// TIA Portal V18 export
FUNCTION_BLOCK "MES Check_fb"   // FB110, LAD
{ S7_Optimized_Access := 'TRUE' }
// stored: AutoNumber false, MemoryReserve 100, SetENOAutomatically false
   VAR_INPUT
      i_AlwaysTrue : Bool;
      i_MESOnlineOffline : Bool;
      i_CheckRequest : Bool;
      i_ResultRequest : Bool;
      i_Reset : Bool;
      i_CheckTimeOut : DInt := 10000;
      i_ResultTimeOut : DInt := 10000;
      i_Status : Int;
   END_VAR
   VAR_OUTPUT
      o_CheckTimeOut : Bool;
      o_ResultTimeOut : Bool;
   END_VAR
   VAR_IN_OUT
      ioPLC_MESCheckReq : Bool;
      ioPLC_MESResultReq : Bool;
      ioMES_PLCChecOK : Bool;
      ioMES_PLCChecNG : Bool;
      ioMES_PLCChecDone : Bool;
      ioMES_PLCResultOK : Bool;
      ioMES_PLCResultNG : Bool;
      ioMES_PLCResultDone : Bool;
      ioProductStatus : Int;
   END_VAR
   VAR
      CheckStep : Int;
      ResultStep : Int;
      CheckTimeOut : TON_TIME;
      ResultTimeOut { S7_SetPoint := 'True'} : TON_TIME;
      Pls : Array[0..20] of Bool;
   END_VAR
   VAR_TEMP   // added for the SCL form of the ladder/FBD networks
      _w1 : Bool;
      _w2 : Bool;
      _w3 : Bool;
      _w4 : Bool;
      _w5 : Bool;
      _w6 : Bool;
      _w7 : Bool;
   END_VAR
BEGIN

REGION Network 1: MES Check In Start
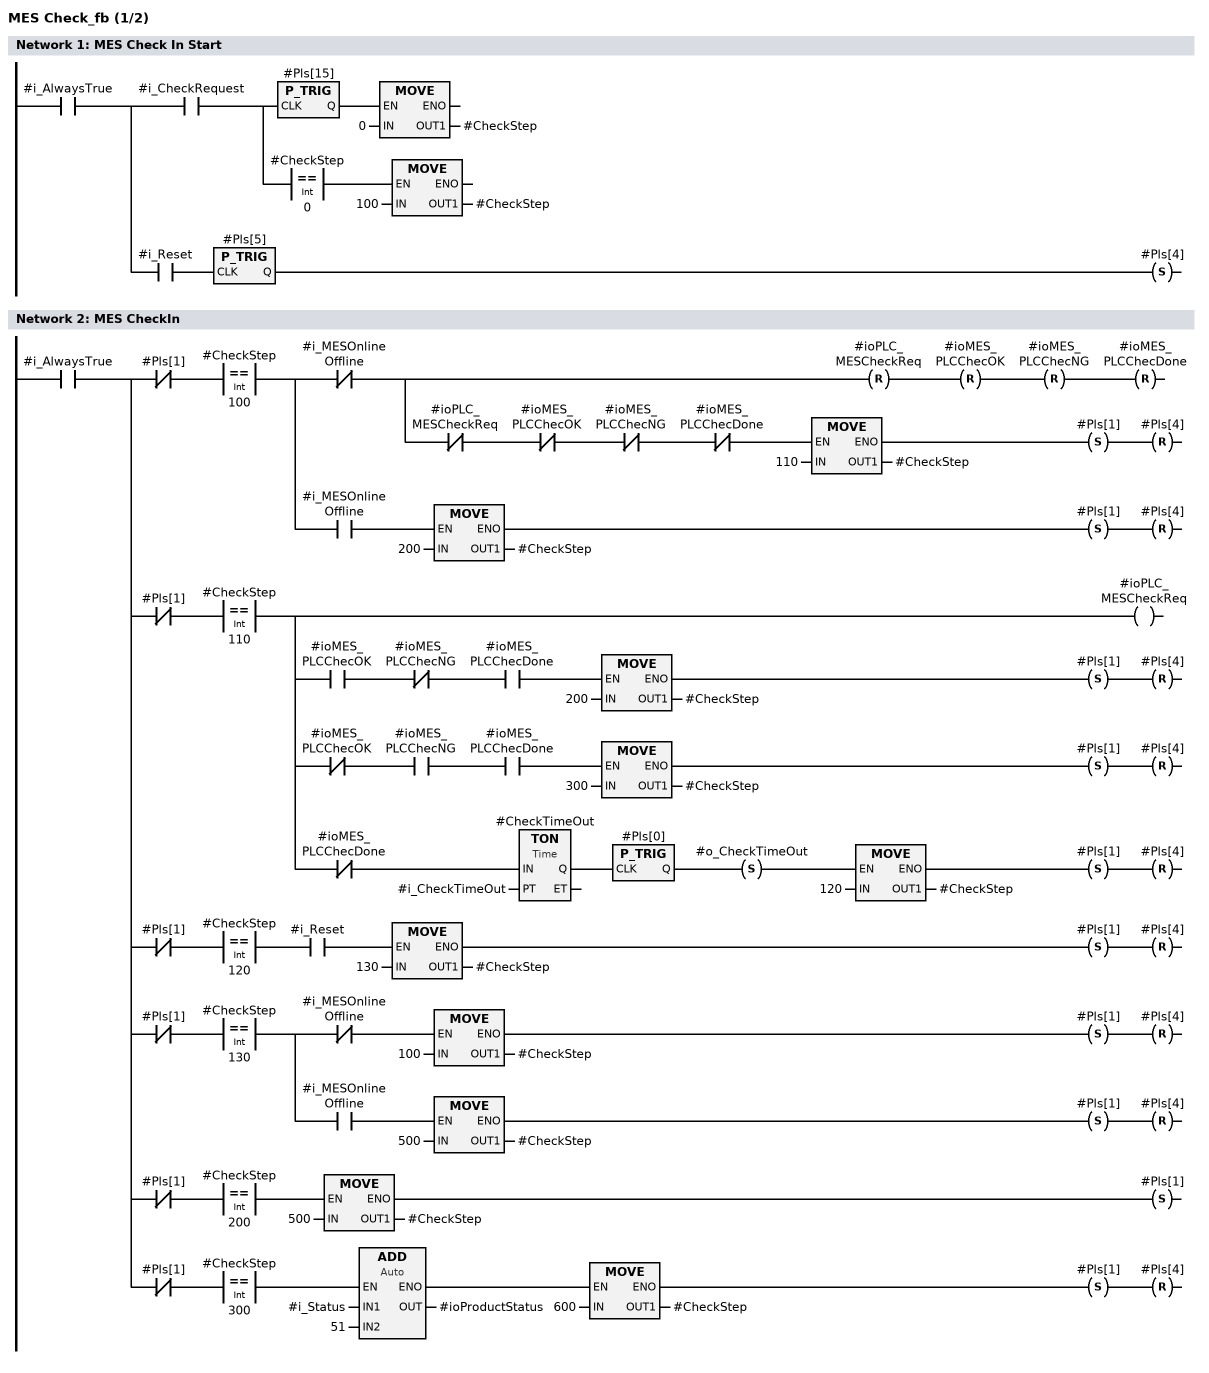
   RUNG wire#powerrail
      Contact( #i_AlwaysTrue )
      wire#w1
      Contact( #i_CheckRequest )
      wire#w2
      P_Trig( #Pls[15] )
      Move(in := 0, out1 => #CheckStep)
   END_RUNG
   RUNG wire#w2
      { S7_Templates := "SrcType := Int" } EQ_Contact(in1 := #CheckStep, in2 := 0)
      Move(in := 100, out1 => #CheckStep)
   END_RUNG
   RUNG wire#w1
      Contact( #i_Reset )
      P_Trig( #Pls[5] )
      S_Coil( #Pls[4] )
   END_RUNG
   // the same network as SCL:
   #_w1 := #i_AlwaysTrue AND #i_CheckRequest;
   #_w2 := #_w1 AND NOT #Pls[15];   // rising edge
   #Pls[15] := #_w1;
   IF #_w2 THEN #CheckStep := 0; END_IF;
   IF #_w1 AND (#CheckStep = 0) THEN #CheckStep := 100; END_IF;
   #_w3 := #i_AlwaysTrue AND #i_Reset;
   #_w4 := #_w3 AND NOT #Pls[5];   // rising edge
   #Pls[5] := #_w3;
   IF #_w4 THEN #Pls[4] := TRUE; END_IF;
END_REGION

REGION Network 2: MES CheckIn
   RUNG wire#powerrail
      Contact( #i_AlwaysTrue )
      wire#w1
      I_Contact( #Pls[1] )
      { S7_Templates := "SrcType := Int" } EQ_Contact(in1 := #CheckStep, in2 := 100)
      wire#w2
      I_Contact( #i_MESOnlineOffline )
      wire#w3
      R_Coil( #ioPLC_MESCheckReq )
      R_Coil( #ioMES_PLCChecOK )
      R_Coil( #ioMES_PLCChecNG )
      R_Coil( #ioMES_PLCChecDone )
   END_RUNG
   RUNG wire#w3
      I_Contact( #ioPLC_MESCheckReq )
      I_Contact( #ioMES_PLCChecOK )
      I_Contact( #ioMES_PLCChecNG )
      I_Contact( #ioMES_PLCChecDone )
      Move(in := 110, out1 => #CheckStep)
      S_Coil( #Pls[1] )
      R_Coil( #Pls[4] )
   END_RUNG
   RUNG wire#w2
      Contact( #i_MESOnlineOffline )
      Move(in := 200, out1 => #CheckStep)
      S_Coil( #Pls[1] )
      R_Coil( #Pls[4] )
   END_RUNG
   RUNG wire#w1
      I_Contact( #Pls[1] )
      { S7_Templates := "SrcType := Int" } EQ_Contact(in1 := #CheckStep, in2 := 110)
      wire#w4
      Coil( #ioPLC_MESCheckReq )
   END_RUNG
   RUNG wire#w4
      Contact( #ioMES_PLCChecOK )
      I_Contact( #ioMES_PLCChecNG )
      Contact( #ioMES_PLCChecDone )
      Move(in := 200, out1 => #CheckStep)
      S_Coil( #Pls[1] )
      R_Coil( #Pls[4] )
   END_RUNG
   RUNG wire#w4
      I_Contact( #ioMES_PLCChecOK )
      Contact( #ioMES_PLCChecNG )
      Contact( #ioMES_PLCChecDone )
      Move(in := 300, out1 => #CheckStep)
      S_Coil( #Pls[1] )
      R_Coil( #Pls[4] )
   END_RUNG
   RUNG wire#w4
      I_Contact( #ioMES_PLCChecDone )
      { S7_Templates := "time_type := Time" } #CheckTimeOut.TON(pt := #i_CheckTimeOut, et =>)
      P_Trig( #Pls[0] )
      S_Coil( #o_CheckTimeOut )
      Move(in := 120, out1 => #CheckStep)
      S_Coil( #Pls[1] )
      R_Coil( #Pls[4] )
   END_RUNG
   RUNG wire#w1
      I_Contact( #Pls[1] )
      { S7_Templates := "SrcType := Int" } EQ_Contact(in1 := #CheckStep, in2 := 120)
      Contact( #i_Reset )
      Move(in := 130, out1 => #CheckStep)
      S_Coil( #Pls[1] )
      R_Coil( #Pls[4] )
   END_RUNG
   RUNG wire#w1
      I_Contact( #Pls[1] )
      { S7_Templates := "SrcType := Int" } EQ_Contact(in1 := #CheckStep, in2 := 130)
      wire#w5
      I_Contact( #i_MESOnlineOffline )
      Move(in := 100, out1 => #CheckStep)
      S_Coil( #Pls[1] )
      R_Coil( #Pls[4] )
   END_RUNG
   RUNG wire#w5
      Contact( #i_MESOnlineOffline )
      Move(in := 500, out1 => #CheckStep)
      S_Coil( #Pls[1] )
      R_Coil( #Pls[4] )
   END_RUNG
   RUNG wire#w1
      I_Contact( #Pls[1] )
      { S7_Templates := "SrcType := Int" } EQ_Contact(in1 := #CheckStep, in2 := 200)
      Move(in := 500, out1 => #CheckStep)
      S_Coil( #Pls[1] )
   END_RUNG
   RUNG wire#w1
      I_Contact( #Pls[1] )
      { S7_Templates := "SrcType := Int" } EQ_Contact(in1 := #CheckStep, in2 := 300)
      Add(in1 := #i_Status, in2 := 51, out => #ioProductStatus)
      Move(in := 600, out1 => #CheckStep)
      S_Coil( #Pls[1] )
      R_Coil( #Pls[4] )
   END_RUNG
   // the same network as SCL:
   #_w1 := #i_AlwaysTrue AND NOT #Pls[1] AND (#CheckStep = 100);
   #_w2 := #_w1 AND NOT #i_MESOnlineOffline;
   IF #_w2 THEN
       #ioPLC_MESCheckReq := FALSE;
       #ioMES_PLCChecOK := FALSE;
       #ioMES_PLCChecNG := FALSE;
       #ioMES_PLCChecDone := FALSE;
   END_IF;
   IF #_w2 AND NOT #ioPLC_MESCheckReq AND NOT #ioMES_PLCChecOK AND NOT #ioMES_PLCChecNG AND NOT #ioMES_PLCChecDone THEN
       #CheckStep := 110;
       #Pls[1] := TRUE;
       #Pls[4] := FALSE;
   END_IF;
   IF #_w1 AND #i_MESOnlineOffline THEN
       #CheckStep := 200;
       #Pls[1] := TRUE;
       #Pls[4] := FALSE;
   END_IF;
   #ioPLC_MESCheckReq := #i_AlwaysTrue AND NOT #Pls[1] AND (#CheckStep = 110);
   IF #ioPLC_MESCheckReq AND #ioMES_PLCChecOK AND NOT #ioMES_PLCChecNG AND #ioMES_PLCChecDone THEN
       #CheckStep := 200;
       #Pls[1] := TRUE;
       #Pls[4] := FALSE;
   END_IF;
   IF #ioPLC_MESCheckReq AND NOT #ioMES_PLCChecOK AND #ioMES_PLCChecNG AND #ioMES_PLCChecDone THEN
       #CheckStep := 300;
       #Pls[1] := TRUE;
       #Pls[4] := FALSE;
   END_IF;
   #CheckTimeOut(IN := #ioPLC_MESCheckReq AND NOT #ioMES_PLCChecDone, PT := #i_CheckTimeOut);   // TON
   #_w3 := #CheckTimeOut.Q AND NOT #Pls[0];   // rising edge
   #Pls[0] := #CheckTimeOut.Q;
   IF #_w3 THEN
       #o_CheckTimeOut := TRUE;
       #CheckStep := 120;
       #Pls[1] := TRUE;
       #Pls[4] := FALSE;
   END_IF;
   #_w4 := #i_AlwaysTrue AND NOT #Pls[1] AND (#CheckStep = 120) AND #i_Reset;
   IF #_w4 THEN
       #CheckStep := 130;
       #Pls[1] := TRUE;
       #Pls[4] := FALSE;
   END_IF;
   #_w5 := #i_AlwaysTrue AND NOT #Pls[1] AND (#CheckStep = 130);
   IF #_w5 AND NOT #i_MESOnlineOffline THEN
       #CheckStep := 100;
       #Pls[1] := TRUE;
       #Pls[4] := FALSE;
   END_IF;
   IF #_w5 AND #i_MESOnlineOffline THEN
       #CheckStep := 500;
       #Pls[1] := TRUE;
       #Pls[4] := FALSE;
   END_IF;
   #_w6 := #i_AlwaysTrue AND NOT #Pls[1] AND (#CheckStep = 200);
   IF #_w6 THEN
       #CheckStep := 500;
       #Pls[1] := TRUE;
   END_IF;
   IF #i_AlwaysTrue AND NOT #Pls[1] AND (#CheckStep = 300) THEN #ioProductStatus := #i_Status + 51; END_IF;
   #_w7 := #i_AlwaysTrue AND NOT #Pls[1] AND (#CheckStep = 300);
   IF #_w7 THEN
       #CheckStep := 600;
       #Pls[1] := TRUE;
       #Pls[4] := FALSE;
   END_IF;
END_REGION

REGION Network 4: MES Check Out Start
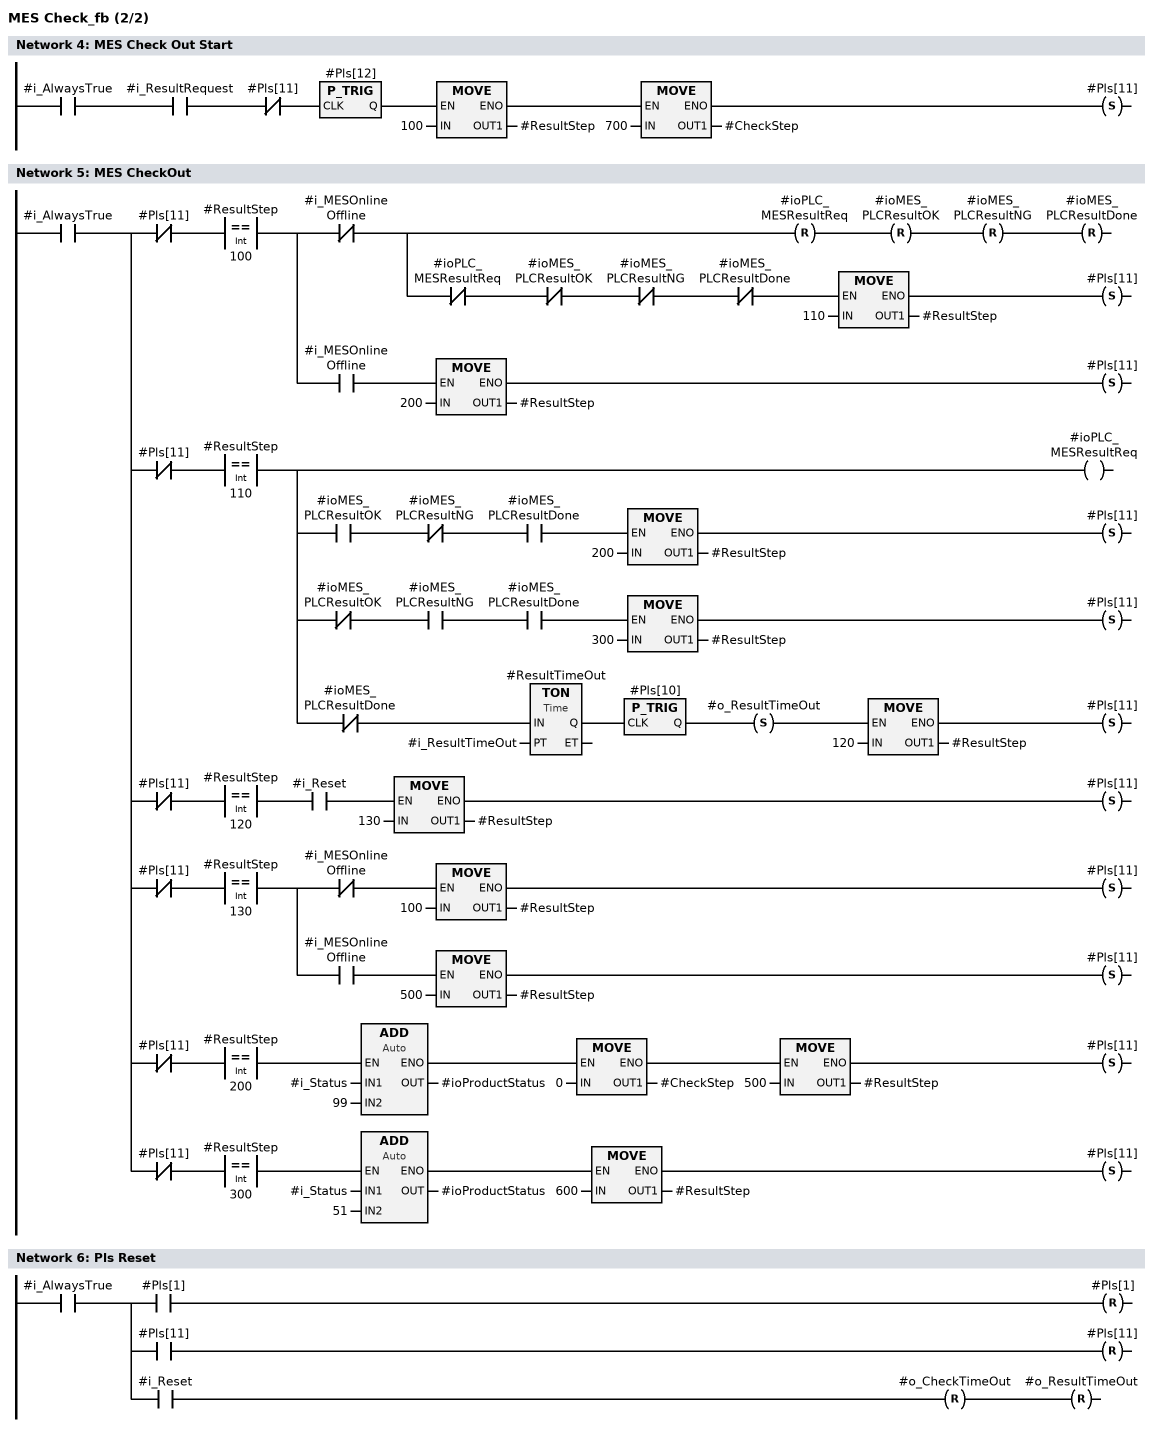
   RUNG wire#powerrail
      Contact( #i_AlwaysTrue )
      Contact( #i_ResultRequest )
      I_Contact( #Pls[11] )
      P_Trig( #Pls[12] )
      Move(in := 100, out1 => #ResultStep)
      Move(in := 700, out1 => #CheckStep)
      S_Coil( #Pls[11] )
   END_RUNG
   // the same network as SCL:
   #_w1 := #i_AlwaysTrue AND #i_ResultRequest AND NOT #Pls[11];
   #_w2 := #_w1 AND NOT #Pls[12];   // rising edge
   #Pls[12] := #_w1;
   IF #_w2 THEN
       #ResultStep := 100;
       #CheckStep := 700;
       #Pls[11] := TRUE;
   END_IF;
END_REGION

REGION Network 5: MES CheckOut
   RUNG wire#powerrail
      Contact( #i_AlwaysTrue )
      wire#w1
      I_Contact( #Pls[11] )
      { S7_Templates := "SrcType := Int" } EQ_Contact(in1 := #ResultStep, in2 := 100)
      wire#w2
      I_Contact( #i_MESOnlineOffline )
      wire#w3
      R_Coil( #ioPLC_MESResultReq )
      R_Coil( #ioMES_PLCResultOK )
      R_Coil( #ioMES_PLCResultNG )
      R_Coil( #ioMES_PLCResultDone )
   END_RUNG
   RUNG wire#w3
      I_Contact( #ioPLC_MESResultReq )
      I_Contact( #ioMES_PLCResultOK )
      I_Contact( #ioMES_PLCResultNG )
      I_Contact( #ioMES_PLCResultDone )
      Move(in := 110, out1 => #ResultStep)
      S_Coil( #Pls[11] )
   END_RUNG
   RUNG wire#w2
      Contact( #i_MESOnlineOffline )
      Move(in := 200, out1 => #ResultStep)
      S_Coil( #Pls[11] )
   END_RUNG
   RUNG wire#w1
      I_Contact( #Pls[11] )
      { S7_Templates := "SrcType := Int" } EQ_Contact(in1 := #ResultStep, in2 := 110)
      wire#w4
      Coil( #ioPLC_MESResultReq )
   END_RUNG
   RUNG wire#w4
      Contact( #ioMES_PLCResultOK )
      I_Contact( #ioMES_PLCResultNG )
      Contact( #ioMES_PLCResultDone )
      Move(in := 200, out1 => #ResultStep)
      S_Coil( #Pls[11] )
   END_RUNG
   RUNG wire#w4
      I_Contact( #ioMES_PLCResultOK )
      Contact( #ioMES_PLCResultNG )
      Contact( #ioMES_PLCResultDone )
      Move(in := 300, out1 => #ResultStep)
      S_Coil( #Pls[11] )
   END_RUNG
   RUNG wire#w4
      I_Contact( #ioMES_PLCResultDone )
      { S7_Templates := "time_type := Time" } #ResultTimeOut.TON(pt := #i_ResultTimeOut, et =>)
      P_Trig( #Pls[10] )
      S_Coil( #o_ResultTimeOut )
      Move(in := 120, out1 => #ResultStep)
      S_Coil( #Pls[11] )
   END_RUNG
   RUNG wire#w1
      I_Contact( #Pls[11] )
      { S7_Templates := "SrcType := Int" } EQ_Contact(in1 := #ResultStep, in2 := 120)
      Contact( #i_Reset )
      Move(in := 130, out1 => #ResultStep)
      S_Coil( #Pls[11] )
   END_RUNG
   RUNG wire#w1
      I_Contact( #Pls[11] )
      { S7_Templates := "SrcType := Int" } EQ_Contact(in1 := #ResultStep, in2 := 130)
      wire#w5
      I_Contact( #i_MESOnlineOffline )
      Move(in := 100, out1 => #ResultStep)
      S_Coil( #Pls[11] )
   END_RUNG
   RUNG wire#w5
      Contact( #i_MESOnlineOffline )
      Move(in := 500, out1 => #ResultStep)
      S_Coil( #Pls[11] )
   END_RUNG
   RUNG wire#w1
      I_Contact( #Pls[11] )
      { S7_Templates := "SrcType := Int" } EQ_Contact(in1 := #ResultStep, in2 := 200)
      Add(in1 := #i_Status, in2 := 99, out => #ioProductStatus)
      Move(in := 0, out1 => #CheckStep)
      Move(in := 500, out1 => #ResultStep)
      S_Coil( #Pls[11] )
   END_RUNG
   RUNG wire#w1
      I_Contact( #Pls[11] )
      { S7_Templates := "SrcType := Int" } EQ_Contact(in1 := #ResultStep, in2 := 300)
      Add(in1 := #i_Status, in2 := 51, out => #ioProductStatus)
      Move(in := 600, out1 => #ResultStep)
      S_Coil( #Pls[11] )
   END_RUNG
   // the same network as SCL:
   #_w1 := #i_AlwaysTrue AND NOT #Pls[11] AND (#ResultStep = 100);
   #_w2 := #_w1 AND NOT #i_MESOnlineOffline;
   IF #_w2 THEN
       #ioPLC_MESResultReq := FALSE;
       #ioMES_PLCResultOK := FALSE;
       #ioMES_PLCResultNG := FALSE;
       #ioMES_PLCResultDone := FALSE;
   END_IF;
   IF #_w2 AND NOT #ioPLC_MESResultReq AND NOT #ioMES_PLCResultOK AND NOT #ioMES_PLCResultNG AND NOT #ioMES_PLCResultDone THEN
       #ResultStep := 110;
       #Pls[11] := TRUE;
   END_IF;
   IF #_w1 AND #i_MESOnlineOffline THEN
       #ResultStep := 200;
       #Pls[11] := TRUE;
   END_IF;
   #ioPLC_MESResultReq := #i_AlwaysTrue AND NOT #Pls[11] AND (#ResultStep = 110);
   IF #ioPLC_MESResultReq AND #ioMES_PLCResultOK AND NOT #ioMES_PLCResultNG AND #ioMES_PLCResultDone THEN
       #ResultStep := 200;
       #Pls[11] := TRUE;
   END_IF;
   IF #ioPLC_MESResultReq AND NOT #ioMES_PLCResultOK AND #ioMES_PLCResultNG AND #ioMES_PLCResultDone THEN
       #ResultStep := 300;
       #Pls[11] := TRUE;
   END_IF;
   #ResultTimeOut(IN := #ioPLC_MESResultReq AND NOT #ioMES_PLCResultDone, PT := #i_ResultTimeOut);   // TON
   #_w3 := #ResultTimeOut.Q AND NOT #Pls[10];   // rising edge
   #Pls[10] := #ResultTimeOut.Q;
   IF #_w3 THEN
       #o_ResultTimeOut := TRUE;
       #ResultStep := 120;
       #Pls[11] := TRUE;
   END_IF;
   #_w4 := #i_AlwaysTrue AND NOT #Pls[11] AND (#ResultStep = 120) AND #i_Reset;
   IF #_w4 THEN
       #ResultStep := 130;
       #Pls[11] := TRUE;
   END_IF;
   #_w5 := #i_AlwaysTrue AND NOT #Pls[11] AND (#ResultStep = 130);
   IF #_w5 AND NOT #i_MESOnlineOffline THEN
       #ResultStep := 100;
       #Pls[11] := TRUE;
   END_IF;
   IF #_w5 AND #i_MESOnlineOffline THEN
       #ResultStep := 500;
       #Pls[11] := TRUE;
   END_IF;
   IF #i_AlwaysTrue AND NOT #Pls[11] AND (#ResultStep = 200) THEN
       #ioProductStatus := #i_Status + 99;
       #CheckStep := 0;
   END_IF;
   #_w6 := #i_AlwaysTrue AND NOT #Pls[11] AND (#ResultStep = 200);
   IF #_w6 THEN
       #ResultStep := 500;
       #Pls[11] := TRUE;
   END_IF;
   IF #i_AlwaysTrue AND NOT #Pls[11] AND (#ResultStep = 300) THEN #ioProductStatus := #i_Status + 51; END_IF;
   #_w7 := #i_AlwaysTrue AND NOT #Pls[11] AND (#ResultStep = 300);
   IF #_w7 THEN
       #ResultStep := 600;
       #Pls[11] := TRUE;
   END_IF;
END_REGION

REGION Network 6: Pls Reset
   RUNG wire#powerrail
      Contact( #i_AlwaysTrue )
      wire#w1
      Contact( #Pls[1] )
      R_Coil( #Pls[1] )
   END_RUNG
   RUNG wire#w1
      Contact( #Pls[11] )
      R_Coil( #Pls[11] )
   END_RUNG
   RUNG wire#w1
      Contact( #i_Reset )
      R_Coil( #o_CheckTimeOut )
      R_Coil( #o_ResultTimeOut )
   END_RUNG
   // the same network as SCL:
   IF #i_AlwaysTrue AND #Pls[1] THEN #Pls[1] := FALSE; END_IF;
   IF #i_AlwaysTrue AND #Pls[11] THEN #Pls[11] := FALSE; END_IF;
   IF #i_AlwaysTrue AND #i_Reset THEN
       #o_CheckTimeOut := FALSE;
       #o_ResultTimeOut := FALSE;
   END_IF;
END_REGION
END_FUNCTION_BLOCK
